// TIA Portal V17 export
// export: Created 2025-06-26T06:49:31.0526413Z, ExportSetting WithDefaults, DisplayName Totally Integrated Automation Portal, DisplayVersion V17 Update 8, DisplayName TIA Portal Openness, DisplayVersion V17 Update 8, DisplayName TIA Portal Version Control Interface, DisplayVersion V17, DisplayName STEP 7 Professional, DisplayVersion V17 Update 8, DisplayName STEP 7 Safety, DisplayVersion V17 Update 6, DisplayName WinCC Advanced, DisplayVersion V17 Update 8
TYPE "stPurgeControl"
// stored: IsFailsafeCompliant false
   STRUCT
      nPurgeCycles : Int;   // [1] How many purge cycles to run
      nPurgeCyclesRemaining : Int;   // [1] How many purge cycles are left to run
      bEnable : Bool;   // 1 = enable from HMI, 0 = disable from HMI
      bFault : Bool;   // 1 = controller fault, 0 = ok
      bReset : Bool;   // 1 = reset controller, 0 = do nothing
      bPurging : Bool;   // 1 = purging, 0 = not purging
      bSpinning : Bool;   // 1 = spinning, 0 = not spinning
      bDone : Bool;   // 1 = purge cycle completed, 0 = not completed
      nMode : USInt;   // 0 = off, 1 = auto, 2 = manual
      fSpinOut : Real;   // [rpm] Spin setpoint (includes ramping)
      Purge : Struct
         nPurgeType : USInt;   // 0 = timer, 1 = delta P, 2 = timer or delta P, 3 = no purge
         tPurgeTime : Time;   // [s] How long to open the purge valves
         fPurgeDeltaP : Real;   // [kPa] Lower limit for pump delta P
      END_STRUCT;
      Spin : Struct
         tSpinTime : Time;   // [s] How long to spin for
         fSpinSpeed : Real;   // [rpm] Spin speed
         fSpinRamp : Real;   // [rpm/s] Spin ramp
      END_STRUCT;
   END_STRUCT;
END_TYPE
